Universal Robots PolyScope program: d02_replug.urp

Program d02_replug (installation=default directory=/programs createdIn=5.9.1.1031110 lastSavedIn=5.9.1.1031110 robotSerialNumber=20195501059)
Calibrated DH parameters: a=[0.000146, -0.418764, -0.053981, 0.000058, -0.000023, 0]; d=[0.162545, 37.319448, -206.067439, 168.881546, 0.09955, 0.099464]; alpha=[1.57004, -0.001979, 0.002304, 1.570607, -1.57066, 0]; deltaTheta=[0, -0.174616, -1.258233, 1.432844, -0.000001, 0]
Robot Program (runOnlyOnce=true)
  URCap Insertion (Robotiq_Copilot, Robotiq Inc.) dataModel(NodeInitializedKey=true)
    URCap Zero FT Sensor (Robotiq_Copilot, Robotiq Inc.) dataModel(NodeInitializedKey=true, WaitForSteadyWrenchOptionKey=false)
    URCap Linear (Robotiq_Copilot, Robotiq Inc.) dataModel(NodeInitializedKey=true, fb_exit_insertion=false, fb_max_distance=50.0, fb_speed=10.0, fb_force=40.0, fbDirection=X-); state(isChildrenLocked=true)
      URCap On error (Robotiq_Copilot, Robotiq Inc.)
        'Sequence if maximum distance is reached'
        Halt
    URCap Gripper (Robotiq_Grippers, Robotiq Inc.) dataModel(position=65.0, force=100.0, speed=100.0, positionInDouble=65.0, forceInDouble=100.0, speedInDouble=100.0, slaveIds=[9], blocking=true)
    MoveL speed 250 mm/s, acceleration 1200 mm/s^2 (useActiveTCP=true) feature=Base
      MoveDirectionNode (selectedDirection=ZMinus) feature=Joint_6_name
        Until DISTANCE (allowActions=false deceleration=3 distanceNodeType=STOP) Distance=0.025; motionParameters(blendRadius=0)
